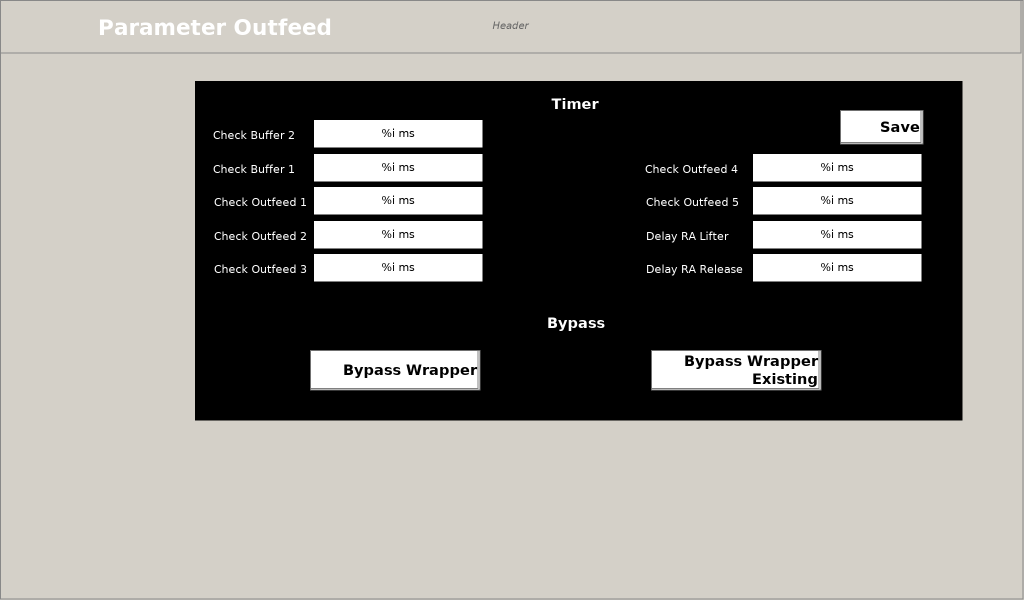
VISUALIZATION MOutfeed  // 1024x600
    Frame (0,-2 1021x55)
        shows Header()
    Label (95,15 250x25), "Parameter Outfeed"
    RoundedRectangle (195,81 767x339)
    Label (223,84 704x40), "Timer"
    Label (210,118 91x35), "Check Buffer 2"
    RoundedRectangle (313,119 170x29), "%i ms", text variable: HMI_GVL.Tmr_PalletBuffer2
        OnMouseClick: write the text variable via Default
    Button (840,110 83x34), "Save", image: VisuSymbols.Symbols.Save
        tap InputOutput_GVL.TestMode[100]
    Label (210,152 91x35), "Check Buffer 1"
    RoundedRectangle (313,153 170x29), "%i ms", text variable: HMI_GVL.Tmr_PalletBuffer1
        OnMouseClick: write the text variable via Default
    Label (642,152 102x35), "Check Outfeed 4"
    RoundedRectangle (752,153 170x29), "%i ms", text variable: HMI_GVL.Tmr_PalletOutfeed4
        OnMouseClick: write the text variable via Default
    Label (211,185 102x35), "Check Outfeed 1"
    RoundedRectangle (313,186 170x29), "%i ms", text variable: HMI_GVL.Tmr_PalletOutfeed1
        OnMouseClick: write the text variable via Default
    Label (643,185 102x35), "Check Outfeed 5"
    RoundedRectangle (752,186 170x29), "%i ms", text variable: HMI_GVL.Tmr_PalletOutfeed5
        OnMouseClick: write the text variable via Default
    Label (211,219 100x35), "Check Outfeed 2"
    RoundedRectangle (313,220 170x29), "%i ms", text variable: HMI_GVL.Tmr_PalletOutfeed2
        OnMouseClick: write the text variable via Default
    Label (643,219 102x35), "Delay RA Lifter"
    RoundedRectangle (752,220 170x29), "%i ms", text variable: HMI_GVL.Tmr_PalletRA
        OnMouseClick: write the text variable via Default
    Label (211,252 100x35), "Check Outfeed 3"
    RoundedRectangle (313,253 170x29), "%i ms", text variable: HMI_GVL.Tmr_PalletOutfeed3
        OnMouseClick: write the text variable via Default
    Label (643,252 102x35), "Delay RA Release"
    RoundedRectangle (752,253 170x29), "%i ms", text variable: HMI_GVL.TmrDelay_PalletRA
        OnMouseClick: write the text variable via Default
    Label (224,303 704x40), "Bypass"
    Button (651,350 170x40), "Bypass Wrapper Existing", colour toggle: HMI_GVL.BypassWrapperExisting, image: VisuSymbols.Symbols.Lock
        toggle HMI_GVL.BypassWrapperExisting
    Button (310,350 170x40), "Bypass Wrapper", colour toggle: HMI_GVL.BypassWrapper, image: VisuSymbols.Symbols.Lock
        toggle HMI_GVL.BypassWrapper
END_VISUALIZATION

(* stored: Version 1.1.0.1, ProductVersion 3.1.4024.12
   Visu MOutfeed: Id {951db375-603f-45c4-bb04-335870b72e63} *)
